// TIA Portal project "SiemensS7-modbus-TCPIP-server" (V16)

(* hardware
DEVICE "S71500/ET200MP station_1"  S7-1500 station
   slot 0: "Rail_0"  Rack  6ES7 590-1***0-0AA0
   slot 1: "PLC_1"  CPU 1512C-1 PN  6ES7 512-1CK01-0AB0  V2.8
      slot 3: "CPU display_1"  6ES7591-1AA00-0AA0
      slot 32768: "PROFINET interface_1"  X1
         slot 32769: "Port_1"  X1 P1
         slot 32770: "Port_2"  X1 P2
      slot 34817: "Virtual CP interface port_1"  Virtual CP interface port  Virtual CP interface port
*)

// ===== PLC "PLC_1"  CPU 1512C-1 PN =====

DATA_BLOCK "Modbus_parameters"   // DB2
{ S7_Optimized_Access := 'FALSE' }
VERSION : 0.1
   VAR
      NDR : Bool;
      DR : Bool;
      ERROR : Bool;
      STATUS : Word;
      CONNECT : TCON_IP_v4;
   END_VAR
BEGIN
   CONNECT.InterfaceId := 64;
   CONNECT.ID := 16#1;
   CONNECT.LocalPort := 502;
END_DATA_BLOCK

DATA_BLOCK "Modbus_data"   // DB3
{ S7_Optimized_Access := 'FALSE' }
VERSION : 0.1
   VAR
      DATA_1 : Array[0..4] of Int;
      DATA_2 : Array[0..2] of Int;
   END_VAR
BEGIN
END_DATA_BLOCK

ORGANIZATION_BLOCK "Main"   // OB1, LAD, ProgramCycle
TITLE = "Main Program Sweep (Cycle)"
{ S7_Optimized_Access := 'TRUE' }
VERSION : 0.1
   VAR_INPUT
      Initial_Call : Bool;   // Initial call of this OB
      Remanence : Bool;   // =True, if remanent data are available
   END_VAR
BEGIN

REGION Network 1
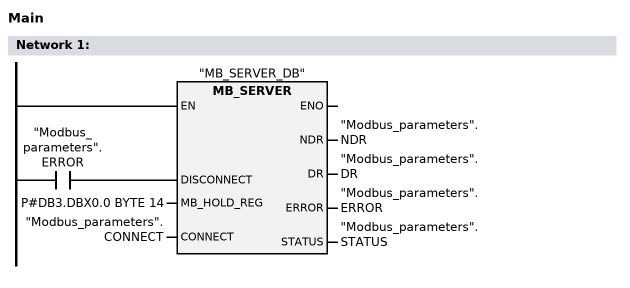
   "MB_SERVER_DB"(DISCONNECT := "Modbus_parameters".ERROR,   // MB_SERVER
                  MB_HOLD_REG := P#DB3.DBX0.0 BYTE 14,
                  CONNECT := "Modbus_parameters".CONNECT,
                  NDR => "Modbus_parameters".NDR,
                  DR => "Modbus_parameters".DR,
                  ERROR => "Modbus_parameters".ERROR,
                  STATUS => "Modbus_parameters".STATUS);
END_REGION
END_ORGANIZATION_BLOCK